// TIA Portal V19 export
FUNCTION "FC_FW_Auftrag_Step4_NB" : Void   // FC184, LAD
TITLE = Schritt WR02 -> CM03
{ S7_Optimized_Access := 'TRUE' }
// Ältesten Warenträger in WR02 suchen und nach CM03 transportieren
// stored: AutoNumber false, SetENOAutomatically false
   VAR_INPUT
      Frg_Einfahrt : Bool;
      Frg_Schritt : Bool;
   END_VAR
   VAR_OUTPUT
      nextStep : Bool;
      startStep : Bool;
      parkStep : Bool;
   END_VAR
   VAR_IN_OUT
      Quelle : Int;
      Ziel : Int;
      Positionen : Array[1..30] of "UDT_Auftrag_Pos";
   END_VAR
   VAR_TEMP
      Sperre_Kurz_li : Bool;
      Sperre_Kurz_li_CM01 : Bool;
      Sperre_Kurz_li_CM02 : Bool;
      Sperre_Kurz_re : Bool;
      Sperre_Kurz_re_CM01 : Bool;
      Sperre_Kurz_re_CM02 : Bool;
      Sperre_Lang : Bool;
      Sperre_Lang_CM01 : Bool;
      Sperre_Lang_CM02 : Bool;
      Vorzug : Bool;
      Befehl_ok : Bool;
      tmpQuelle : Int;
      Oldest : Real;
   END_VAR
BEGIN

REGION Network 1 (SCL)
   IF (#Quelle <> 0) AND (#Ziel <> 0) THEN
       #nextStep := #Positionen[#Quelle].Sperre;
       #startStep := NOT #nextStep;
       #Quelle := 0;
       #Ziel := 0;
       RETURN;
   END_IF;

   #Quelle := 0;
   #Ziel := 0;
   #nextStep := FALSE;
   #startStep := FALSE;

   IF NOT #Frg_Einfahrt OR NOT #Frg_Schritt THEN
       #nextStep := TRUE;
       RETURN;
   END_IF;
END_REGION

REGION Network 2 (SCL): Positionen sperren
   //Groß links nicht möglich
   #Positionen[27].CheckSperre := #Positionen[9].Sperre OR (#Positionen[3].Sperre AND #Positionen[15].Sperre);

   //Groß rechts nicht möglich
   #Positionen[28].CheckSperre := #Positionen[10].Sperre OR (#Positionen[4].Sperre AND #Positionen[16].Sperre);

   //kein Platz für Kurz links in CM03
   #Sperre_Kurz_li_CM01 := #Positionen[1].Sperre AND #Positionen[5].Sperre;
   #Sperre_Kurz_li_CM02 := #Positionen[13].Sperre AND #Positionen[17].Sperre;
   #Sperre_Kurz_li := (#Positionen[7].Sperre AND #Positionen[11].Sperre) OR (#Sperre_Kurz_li_CM01 AND #Sperre_Kurz_li_CM02);

   //kein Platz für Kurz rechts in CM03
   #Sperre_Kurz_re_CM01 := #Positionen[2].Sperre AND #Positionen[6].Sperre;
   #Sperre_Kurz_re_CM02 := #Positionen[14].Sperre AND #Positionen[18].Sperre;
   #Sperre_Kurz_re := (#Positionen[8].Sperre AND #Positionen[12].Sperre) OR (#Sperre_Kurz_re_CM01 AND #Sperre_Kurz_re_CM02);

   //kein Platz für Lang in CM03
   #Sperre_Lang_CM01 := ((#Positionen[1].Sperre OR #Positionen[2].Sperre) AND (#Positionen[5].Sperre OR #Positionen[6].Sperre));
   #Sperre_Lang_CM02 := ((#Positionen[13].Sperre OR #Positionen[14].Sperre) AND (#Positionen[17].Sperre OR #Positionen[18].Sperre));
   #Sperre_Lang := ((#Positionen[7].Sperre OR #Positionen[8].Sperre) AND (#Positionen[11].Sperre OR #Positionen[12].Sperre)) OR (#Sperre_Lang_CM01 AND #Sperre_Lang_CM02);

   //Lang in P25 oder
   //kein Platz auf rechter Seite
   //-> P26 sperren
   #Positionen[26].CheckSperre := #Sperre_Kurz_re OR (#Positionen[25].Wt_Typ = "WT_Typ_LS");

   //Lang in P25 und kein Platz für Lang oder
   //kein Platz auf linker Seite
   //-> P25 sperren
   #Positionen[25].CheckSperre := #Sperre_Kurz_li OR ((#Positionen[25].Wt_Typ = "WT_Typ_LS") AND #Sperre_Lang);

   //Lang in P29 oder
   //kein Platz auf rechter Seite
   //-> P30 sperren
   #Positionen[30].CheckSperre := #Sperre_Kurz_re OR (#Positionen[29].Wt_Typ = "WT_Typ_LS");

   //Lang in P29 und kein Platz für Lang oder
   //kein Platz auf linker Seite
   //-> P29 sperren
   #Positionen[29].CheckSperre := #Sperre_Kurz_li OR ((#Positionen[29].Wt_Typ = "WT_Typ_LS") AND #Sperre_Lang);
END_REGION

REGION Network 3 (SCL): Ältesten WT suchen
   //
   #Oldest := 0;
   #tmpQuelle := 0;

   //WR02
   "FC_FW_Auftrag_Suche"(Pos1 := 25,
                         Pos2 := 30,
                         Positionen := #Positionen,
                         Quelle := #tmpQuelle,
                         Oldest := #Oldest);
END_REGION

REGION Network 4 (SCL): Auswertung
   IF #tmpQuelle = 0 THEN
       //kein WT
       #nextStep := TRUE;
       RETURN;
   END_IF;

   IF NOT #Positionen[#tmpQuelle].Fertig THEN
       #parkStep := TRUE;
       RETURN;
   END_IF;

   IF (#tmpQuelle = 27) THEN
       //Gross links
       IF NOT #Positionen[9].Sperre THEN
           "FC_FW_Auftrag_Befehl"(inQuelle := #tmpQuelle,
                                  inZiel := 9,
                                  Befehl_ok => #Befehl_ok,
                                  outQuelle => #Quelle,
                                  outZiel => #Ziel);

           #nextStep := NOT #Befehl_ok;
       ELSE
           #nextStep := TRUE;
       END_IF;
       RETURN;
   END_IF;

   IF (#tmpQuelle = 28) THEN
       //Gross rechts
       IF NOT #Positionen[10].Sperre THEN
           "FC_FW_Auftrag_Befehl"(inQuelle := #tmpQuelle,
                                  inZiel := 10,
                                  Befehl_ok => #Befehl_ok,
                                  outQuelle => #Quelle,
                                  outZiel => #Ziel);

           #nextStep := NOT #Befehl_ok;
       ELSE
           #nextStep := TRUE;
       END_IF;
       RETURN;
   END_IF;

   IF (#Positionen[#tmpQuelle].Wt_Typ = "WT_Typ_LS") AND ((#tmpQuelle = 25) OR (#tmpQuelle = 29)) THEN
       //Lang
       IF NOT #Positionen[11].Sperre AND NOT #Positionen[12].Sperre THEN
           "FC_FW_Auftrag_Befehl"(inQuelle := #tmpQuelle,
                                  inZiel := 11,
                                  Befehl_ok => #Befehl_ok,
                                  outQuelle => #Quelle,
                                  outZiel => #Ziel);

           #nextStep := NOT #Befehl_ok;
       ELSIF NOT #Positionen[7].Sperre AND NOT #Positionen[8].Sperre THEN
           "FC_FW_Auftrag_Befehl"(inQuelle := #tmpQuelle,
                                  inZiel := 7,
                                  Befehl_ok => #Befehl_ok,
                                  outQuelle => #Quelle,
                                  outZiel => #Ziel);

           #nextStep := NOT #Befehl_ok;
       ELSE
           #nextStep := TRUE;
       END_IF;
       RETURN;
   END_IF;

   IF (#tmpQuelle = 25) OR (#tmpQuelle = 29) THEN
       //Kurz links
       #Vorzug := NOT #Positionen[11].Sperre AND NOT #Positionen[12].Sperre AND NOT #Positionen[7].Sperre AND #Positionen[8].Sperre;

       IF NOT #Positionen[11].Sperre AND NOT #Vorzug THEN
           "FC_FW_Auftrag_Befehl"(inQuelle := #tmpQuelle,
                                  inZiel := 11,
                                  Befehl_ok => #Befehl_ok,
                                  outQuelle => #Quelle,
                                  outZiel => #Ziel);

           #nextStep := NOT #Befehl_ok;
       ELSIF NOT #Positionen[7].Sperre THEN
           "FC_FW_Auftrag_Befehl"(inQuelle := #tmpQuelle,
                                  inZiel := 7,
                                  Befehl_ok => #Befehl_ok,
                                  outQuelle => #Quelle,
                                  outZiel => #Ziel);

           #nextStep := NOT #Befehl_ok;
       ELSE
           #nextStep := TRUE;
       END_IF;
       RETURN;
   END_IF;

   IF (#tmpQuelle = 26) OR (#tmpQuelle = 30) THEN
       //Kurz rechts
       #Vorzug := NOT #Positionen[11].Sperre AND NOT #Positionen[12].Sperre AND #Positionen[7].Sperre AND NOT #Positionen[8].Sperre;

       IF NOT #Positionen[12].Sperre AND NOT #Vorzug THEN
           "FC_FW_Auftrag_Befehl"(inQuelle := #tmpQuelle,
                                  inZiel := 12,
                                  Befehl_ok => #Befehl_ok,
                                  outQuelle => #Quelle,
                                  outZiel => #Ziel);

           #nextStep := NOT #Befehl_ok;
       ELSIF NOT #Positionen[8].Sperre THEN
           "FC_FW_Auftrag_Befehl"(inQuelle := #tmpQuelle,
                                  inZiel := 8,
                                  Befehl_ok => #Befehl_ok,
                                  outQuelle => #Quelle,
                                  outZiel => #Ziel);

           #nextStep := NOT #Befehl_ok;
       ELSE
           #nextStep := TRUE;
       END_IF;
       RETURN;
   END_IF;

   //?
   #nextStep := TRUE;
END_REGION
END_FUNCTION
